FUNCTION_BLOCK FB_EffectiveEncoderResolutionDetection EXTENDS FB_Commons
VAR_INPUT
  (*EL1252*)
  bIKp_MarkTrigger01    AT%I* : BOOL;        // First  mark sensor - Trigger
  tIKp_TimeStampPos01   AT%I* : T_DCTIME64;  // First  mark sensor - RisingEdge  @EL1252
  tIKn_TimeStampNeg01   AT%I* : T_DCTIME64;  // First  mark sensor - FallingEdge @EL1252
  bIKp_MarkTrigger02    AT%I* : BOOL;        // Second mark sensor - Trigger
  tIKp_TimeStampPos02   AT%I* : T_DCTIME64;  // Second mark sensor - RisingEdge  @EL1252
  tIKn_TimeStampNeg02   AT%I* : T_DCTIME64;  // Second mark sensor - FallingEdge @EL1252
  nPulse                      : DINT;        // encoder pulse input
  nDisInPulseFilterSz         : UDINT;       // mav filter size for measured distance in encoder steps (from machine) 
    
  // settings
  fCurrentResolution          : LREAL;       // current used resolution (given from machine), encoder step size
  fEncoderPulseDistMin        : LREAL;       // [pulse] defines the min sensor distance in pulse, range minimum
  fEncoderPulseDistMax        : LREAL;       // [pulse] defines the max sensor distance in pulse, range maximum
  fMinMarkLength              : LREAL:=2000; // [um] minimal mark lenght to accept a measurement
  fMaxMarkLength              : LREAL:=6000; // [um] maximal mark lenght to accept a measurement
END_VAR
VAR_OUTPUT
  bUpdate                     : BOOL;        // a valid new measurment
  fDisInPulse                 : LREAL;       // disntance in encoder pulse
END_VAR
VAR
  bInitOk                     : BOOL;        // initialized
   
  fSpeedPulse                 : LREAL;       // current encoder speed [pulse/s]
  fSpeedUm_s                  : LREAL;       // current speed [um/s]
  fbMark1,fbMark2             : RF_TRIG;     // edge detection
  bMeasurementActive          : BOOL;        // a measurement started
  bS1_MarkStarted, bS2_MarkStarted : BOOL;
  nMeasurementCounter         : UDINT;       // counter for measurements
  nCurrentDistActive          : DINT;        // current distance during active measurement
  bVerbose                    : BOOL;
  // errors
  bLower, bHigher, bAborted   : BOOL;        // ui errors
  bMarkInvalidLength_S1, bMarkInvalidLength_S2 : BOOL; // detected marks too short or too long
  nMarkLength_S1, nMarkLength_S2 : UDINT;    // mark length measured in [um]
  
  // time calculations
  tNowDc                      : T_DCTIME64;  // Get Current Timestamp (now
  _fCycleTime                 : LREAL;       // Current cycle time [s]

  // position
  fDistMeasured               : LREAL;       // distance measured [pulse]
  fbFilterMavDisInPulse       : FB_FILTER_MAV; // Moving everage filter
  //fbFilterMavSpeed            : FB_FILTER_MAV; // Moving everage filter
  fAbortDistUm                : LREAL;
  
  // helper measurement
  nPosStart, nPosEnd : DINT;                 // encoder positions detectec (exact by trigger, timestamp and speed based approximation)
  nPosFalling1, nPosFalling2 : DINT;         // exact position in [pulse]
  bRising_S1, bFalling_S1, bRising_S2, bFalling_S2 : BOOL;    // sensor edge detection

END_VAR
VAR CONSTANT
  nC_MinMarkLength            : LREAL := 2_000; // min. mark length in [um]
END_VAR

// check & correct parameter
IF NOT bInitOk THEN RETURN; END_IF;

bUpdate := FALSE;

// time caluclations
tNowDc := F_GetCurDcTaskTime64();                  // current dc time (most accurate time stamp we have)
_fCycleTime := calcCycleTime(tCurrent:=tNowDc);     // calculate cycle time of this fb

// input edge detection
fbMark1(CLK:=bIKp_MarkTrigger01);
fbMark2(CLK:=bIKp_MarkTrigger02);

// track position & speed
position(
  fResolutionInput:=fCurrentResolution, 
  lPosReference:=nPulse, 
  fMasterSpeed=>fSpeedUm_s,    // [um/s]
  fPulseSpeed=>fSpeedPulse,    // [p/s]
);

measure(bUpdate=>bUpdate, fEncoderDistance=>fDistMeasured);
IF bUpdate THEN
  // check range (given from machine)
  bHigher := SEL(fDistMeasured > fEncoderPulseDistMax, FALSE, TRUE);  IF bVerbose AND bHigher THEN LogWarning('Measured distance in pulse LONGER than max range'); END_IF
  bLower  := SEL(fDistMeasured < fEncoderPulseDistMin, FALSE, TRUE);  IF bVerbose AND bLower  THEN LogWarning('Measured distance in pulse SHORTER than min range'); END_IF

  IF NOT bHigher AND NOT bLower THEN  
    // measurement ok
    fbFilterMavDisInPulse(fI_Input:=fDistMeasured, iI_NbInputs:=TO_UINT(LIMIT(1, nDisInPulseFilterSz, fbFilterMavDisInPulse.cL_BUFFER_MAX))); // moving average filter
    fDisInPulse := fbFilterMavDisInPulse.fO_OutputMav;
  END_IF
  
  nMeasurementCounter := (nMeasurementCounter + 1) MOD 1000;  // limit to 0-1000
END_IF

// 
METHOD PRIVATE abortMarkEndSearch : BOOL
VAR_INPUT
  nStart  : DINT;     // pulse
  nEnd    : DINT;     // pulse
END_VAR
VAR
  nDist   : DINT;     // [pulse]
  fDistUm : LREAL;    // um
END_VAR
// pulse elapsed * resolution [um/pulse] => pos in [um]
nDist := ABS(nEnd - nStart);    // distance in pulse (1-2 cycle too late)
fDistUm := nDist * fCurrentResolution;   // distance in [um]  

fAbortDistUm := fMaxMarkLength + (2*_fCycleTime * fSpeedUm_s);

abortMarkEndSearch := fDistUm > fAbortDistUm;
END_METHOD

METHOD PRIVATE calcCycleTime : LREAL
VAR_INPUT
  tCurrent : T_DCTIME64;
END_VAR
VAR_INST
  tLastTimeStamp : T_DCTIME64 := 0;
END_VAR
calcCycleTime := (TO_LREAL(tCurrent) - TO_LREAL(tLastTimeStamp)) * 1E-9;
tLastTimeStamp  := tCurrent;  // memory timestamp
END_METHOD

METHOD PRIVATE checkMarkLength : BOOL
VAR_INPUT
  nRef : DINT;     // pulse
  nOther : DINT;   // pluse
END_VAR
VAR_OUTPUT
  nLen : DINT;     // mark length in pulse
END_VAR
VAR
  fMarkLen : LREAL;  // [um]
END_VAR
IF fCurrentResolution = 0 THEN RETURN; END_IF

// pulse elapsed * resolution [pulse/um] => pos in [um]
nLen := ABS(nOther - nRef);
fMarkLen := nLen * fCurrentResolution;
IF fMarkLen > fMinMarkLength AND fMarkLen < fMaxMarkLength THEN
  // mark within spec
  checkMarkLength := TRUE;
  IF bVerbose THEN LogInfo(F_Concat3('Mark length= ', TO_STRING(fMarkLen), 'um')); END_IF
ELSE
  IF bVerbose THEN LogWarning(F_Concat5('Mark length invalid: ', TO_STRING(fMarkLen), 'um', ' too short or too long', '')); END_IF
END_IF
END_METHOD

METHOD PRIVATE getExactPosition : DINT
VAR_INPUT
  tNow : T_DCTIME64;    // current system time
  nPos : DINT;          // current (encoder) position at the current timestamp
  tEdge : T_DCTIME64;   // detected time
  fSpeed : LREAL;       // current speed
END_VAR
VAR
  fCurrentTimeStamp : LREAL;
  fSensor_TimeStamp : LREAL;
  fDeltaDistance    : LREAL;      // Distance that the substrate moved between the detection and the treatment of the information
END_VAR
IF fCurrentResolution = 0 THEN RETURN; END_IF

// Calculate the original position in our position domain
fCurrentTimeStamp  := (ULINT_TO_LREAL(tNow) - (GVL_WEU.nC_CurrentTimeStampComp * 1_000)) / 1_000_000.0; // [ms]
fSensor_TimeStamp := (ULINT_TO_LREAL(tEdge) - (GVL_WEU.nC_SensorTimeStampComp  * 1_000)) / 1_000_000.0; // [ms]

// Treatment of the information
fDeltaDistance   := (fCurrentTimeStamp - fSensor_TimeStamp) * 0.001 * fSpeed;	      // Distance in pulses that the substrate has traveled between the sensor detection and the PLC treatment
// not conversion to px   nDeltaPosition := FC_LREAL_TO_DINT(fDeltaDistance * (1 / (0.0254 / fCurrentResolution)));   // 1/1px	(* Travel of the substrate between the time of acquisition and the time of treatment
getExactPosition := FC_LREAL_TO_DINT(TO_LREAL(nPos) - fDeltaDistance);
END_METHOD

METHOD Init
Reset();

bInitOk := TRUE;
END_METHOD

METHOD PRIVATE measure
VAR_OUTPUT
  bUpdate : BOOL;
  fEncoderDistance : LREAL;
END_VAR
bUpdate := FALSE;
bRising_S1 := fbMark1.RT;
bRising_S2 := fbMark2.RT;
bFalling_S1 := fbMark1.FT;    // wait on falling edge always 
bFalling_S2 := fbMark2.FT;

IF NOT bMeasurementActive THEN
  
  //-- S1 sensor evaluation (no measurement is active)
  // rising
  IF bRising_S1 AND NOT bS1_MarkStarted THEN
    nPosStart := getExactPosition(tNow:=tNowDc, nPos:=nPulse, tEdge:=tIKp_TimeStampPos01, fSpeed:=fSpeedPulse);
    bS1_MarkStarted := TRUE;
    bAborted := FALSE; bMarkInvalidLength_S1 := FALSE; bMarkInvalidLength_S2 := FALSE;
  END_IF

  // falling (after rising)
  IF bFalling_S1 AND bS1_MarkStarted THEN
    bS1_MarkStarted := FALSE;           // mark done
    nPosFalling1 := getExactPosition(tNow:=tNowDc, nPos:=nPulse, tEdge:=tIKn_TimeStampNeg01, fSpeed:=fSpeedPulse);
  
    IF checkMarkLength( nRef := nPosStart, nOther := nPosFalling1) THEN
      bMeasurementActive := TRUE;           // start measurement after rising&falling edge
    ELSE
      bMarkInvalidLength_S1 := TRUE;
    END_IF

  // abort mark if no falling given
  ELSIF bS1_MarkStarted AND abortMarkEndSearch(nStart:=nPosStart, nEnd:=nPulse) THEN  // abort if max mark length exeeded
    bS1_MarkStarted := FALSE;         // mark done
    bMarkInvalidLength_S1 := TRUE;    // mark end missed (too long?)
    IF bVerbose THEN LogWarning('S1 mark missing end, mark too long, ignore mark'); END_IF
  END_IF
  
ELSE
  
  //-- S2 Second Sensor (Stop) evaluation when measurement is active
  //   only when measurement started and rising within range
  IF (nPulse - nPosStart) >= fEncoderPulseDistMin THEN                  // bigger than minimum pulse (enable sensor 2 detection)
    // rising
    IF bRising_S2 AND NOT bS2_MarkStarted THEN 
      nPosEnd := getExactPosition(tNow:=tNowDc, nPos:=nPulse, tEdge:=tIKp_TimeStampPos02, fSpeed:=fSpeedPulse);    
      bAborted := FALSE; bMarkInvalidLength_S2 := FALSE;
      bS2_MarkStarted := TRUE;  
    END_IF
    
    // falling
    IF bFalling_S2 AND bS2_MarkStarted THEN
      bS2_MarkStarted := FALSE;
      nPosFalling2 := getExactPosition(tNow:=tNowDc, nPos:=nPulse, tEdge:=tIKn_TimeStampNeg02, fSpeed:=fSpeedPulse);  
      
      IF checkMarkLength( nRef := nPosEnd, nOther := nPosFalling2) THEN
        bUpdate := TRUE;
        bMeasurementActive := FALSE;      // stop measurement
      ELSE
        bMarkInvalidLength_S2 := TRUE;
      END_IF

    // abort mark if no falling given
    ELSIF bS2_MarkStarted AND abortMarkEndSearch(nStart:=nPosEnd, nEnd:=nPulse) THEN  // abort if max mark length exeeded
      bS1_MarkStarted := FALSE;         // mark done
      bMarkInvalidLength_S2 := TRUE;    // mark end missed (too long?)
      IF bVerbose THEN LogWarning('S2 mark missing end, mark too long, ignore mark'); END_IF
    END_IF
  
  // abort measurement, no valid mark within max pulse distance
  //       TODO: the nPulse can be 1-2 cycle later than the nPosStart so maybe we should add a marging here to fEncoderPulseDistMax + 1 cycle
  ELSIF ( (nPulse - nPosStart) > (fEncoderPulseDistMax) ) THEN    // bigger than maximum pulse (disable sensor 2 and abort measurement)
    IF bVerbose THEN LogWarning('S2 mark detected too far , ignore measurement'); END_IF
    bAborted := TRUE;                   // abort measurement
    bMeasurementActive := FALSE;        // abort measurement
    bS2_MarkStarted := FALSE;           // mark done
  
  // invalid speed (machine stopped while measuring) ignore any triggers
  ELSIF fSpeedPulse = 0 THEN
    bS1_MarkStarted := bS2_MarkStarted := FALSE;
    bMeasurementActive := FALSE;
	END_IF
  
END_IF

// debug current distance (view)
IF bMeasurementActive THEN nCurrentDistActive := (nPulse - nPosStart); END_IF 

// valid measurment -> update output
IF bUpdate THEN
  fEncoderDistance := nPosEnd-nPosStart;
END_IF
END_METHOD

METHOD PRIVATE position
VAR_INPUT
  lPosReference         : DINT;			                (*Position reference pulse count in [pulse (resolution)]*)
  fResolutionInput      : LREAL := 1;	              (*Encoder resolution in [um/increment]*)
END_VAR
VAR_OUTPUT
  fMasterPosition       : LREAL;                    (*Master position in [um]*)
  fPulsePosition        : LREAL;
  fMasterSpeed          : LREAL;                    (*Master speed in [um/s]*)
  fPulseSpeed           : LREAL;                    (*Pulse speed*)
END_VAR
VAR_INST
  bReset : BOOL;

  lL_Reference_Reg       : DINT := 0;               (*Position reference pulse count register [pulse (resolution)]*)
  fL_Master_Position_Reg : LREAL := 0;	            (*Master position register (last position) [um]*)
  fL_Pulse_Position_Reg  : LREAL := 0;	            (*Master position register (last position) [?]*)
  lL_Delta               : DINT;                    (*Delta of position reference pulses*)
  fDelta : LREAL;
  fb_MavDelta            : FB_FILTER_MAV;           (*Moving everage filter*)

  fL_MasterSpeed_reg     : LREAL;                   (*Speed register [m/s]*)
  fL_PulseSpeed_reg      : LREAL;                   (*Speed [p/s]*)
END_VAR
VAR CONSTANT
  iC_FilterDepth         : UINT := 1;                (*Default filter depth*)
  fC_MinSpeed            : LREAL := 0.02;            (*min speed [m/s]*)
END_VAR
IF _fCycleTime = 0 THEN RETURN; END_IF
IF bReset THEN bReset := FALSE;
  lL_Reference_Reg := lPosReference;
  fL_Master_Position_reg := 0; fL_Pulse_Position_Reg := 0;
  fL_MasterSpeed_reg := 0; fL_PulseSpeed_reg := 0;
END_IF 

lL_Delta:=UDINT_TO_DINT(lPosReference-lL_Reference_Reg);  // DINT because diff correct on wrap over
// filter
fb_MavDelta.fI_Input    := DINT_TO_LREAL(lL_Delta);       // encoder signal jitter filter
fb_MavDelta.iI_NbInputs := iC_FilterDepth;
fb_MavDelta();
fDelta := TO_LREAL(lL_Delta);    //fb_MavDelta.fO_OutputMav  (filtered)

// Position & Speed Calculation 
fMasterPosition := fDelta * fResolutionInput + fL_Master_Position_Reg;
fPulsePosition  := fDelta * 1 + fL_Pulse_Position_Reg;

(*Speed Calculation*)
fMasterSpeed := (fMasterPosition - fL_Master_Position_Reg) * (1 / _fCycleTime);  // um/s      // * 0.000001 um -> m 
IF LrealIsNaN(x:=fMasterSpeed) THEN fMasterSpeed := fL_MasterSpeed_reg; END_IF
fPulseSpeed  := (fPulsePosition - fL_Pulse_Position_Reg) * (1 / _fCycleTime); // * 0.000001;  // um -> 
IF LrealIsNaN(x:=fPulseSpeed) THEN fPulseSpeed := fL_PulseSpeed_reg; END_IF

(*Update Registers*)
lL_Reference_Reg       := lPosReference;
fL_Master_Position_Reg := fMasterPosition; fL_Pulse_Position_Reg := fPulsePosition;
fL_MasterSpeed_reg     := fMasterSpeed; fL_PulseSpeed_reg := fPulseSpeed;
END_METHOD

METHOD PRIVATE Reset
nMeasurementCounter := 0;
END_METHOD

END_FUNCTION_BLOCK

(* stored: Version 1.1.0.1, ProductVersion 3.1.4024.11
   POU FB_EffectiveEncoderResolutionDetection: Id {172ff757-0f60-4a20-baa8-40d4b6b6387f}, SpecialFunc None
   Method abortMarkEndSearch: Id {59de4153-f433-43c2-84a9-02f391a18c25}
   Method calcCycleTime: Id {d0932db0-858d-4f52-84ae-fb96799c2d8c}
   Method checkMarkLength: Id {a7413c46-e6e0-4347-b06a-9059e8a70b2c}
   Method getExactPosition: Id {64c83f4e-2f90-4829-a9ba-519450c0af9d}
   Method Init: Id {ac39b667-8b90-4a38-b9db-5deaa270f17b}
   Method measure: Id {67cbae6f-8d48-4bd4-86d9-cdcb6b146f3f}
   Method position: Id {53e17ab5-9e13-42f7-bcde-c46ddd8bd1ca}
   Method Reset: Id {d5fe1b7c-5060-4be1-aff0-fdec2471f305} *)
